{attribute 'GeneratedUsingTerminal: EK1960-2600-0019'}
{attribute addProperty BoxType "EK1960-2600-0019"}
{attribute addProperty Description "EK1960-2600 TwinSAFE-Compact-Controller (4 x Relay, RJ45)"}
{attribute addProperty Physics "YKY"}
{attribute addProperty Id "Module_1_FSoEModule_1_FSoE_7E6C60DE104Module_2_FSOUTModule_2_FSOUT_E84B1B0028Module_3_FSLOGICModule_3_FSLOGIC_DEAB45222WcStateAT %I*WcState_B516A2644InfoDataAT %I*InfoData_32EB74EA10"}
{attribute addProperty CRC "3135397356"}
{attribute addProperty Size "148"}
TYPE EK1960_BAE25DEC EXTENDS EtcSlaveBoxBase_77A0E4A7 :
STRUCT
	{attribute addProperty Name "Module_1_FSoE"}
	Module_1_FSoE : Module_1_FSoE_7E6C60DE;
	{attribute addProperty Name "Module_2_FSOUT"}
	Module_2_FSOUT : Module_2_FSOUT_E84B1B00;
	{attribute addProperty Name "Module_3_FSLOGIC"}
	Module_3_FSLOGIC : Module_3_FSLOGIC_DEAB4522;
	{attribute addProperty Name "WcState"}
	WcState : WcState_B516A264;
	{attribute addProperty Name "InfoData"}
	InfoData : InfoData_32EB74EA;
END_STRUCT
END_TYPE

(* stored: Version 1.2.0.0, ProductVersion 3.1.4024.11
   DUT EK1960_BAE25DEC: Id {eb8e8251-8c42-4bc4-9596-aa2680afcf71} *)
